(* IEC 61131-3 sources: Idecon_CheckWeigher_WP/03_FC, 6 files *)

(* ---- FC_Idecon_ResetBatch.st ---- *)
// ==============================================================================
// FUNZIONE: FC_Idecon_ResetBatch
// DESCRIZIONE: Resetta statistiche batch su cambio lotto
// INPUT: CurrentBatchCode (STRING[64]) - Codice lotto corrente
// OUTPUT: BatchResetDone (BOOL) - TRUE se reset eseguito
// NOTE: Implementare nel task ciclico monitorando cambio G_Idecon_BatchCode
// ==============================================================================

VAR_INPUT
    CurrentBatchCode : STRING[64];
END_VAR

VAR_OUTPUT
    BatchResetDone : BOOL;
END_VAR

VAR
    PreviousBatchCode : STRING[64];
    CurrentTimestamp_Unix_ms : LINT;
END_VAR

// Get current timestamp (requires SysTicks function or PLC time)
// CurrentTimestamp_Unix_ms := ...;  // Da implementare con funzione di sistema

// Detect batch code change
IF CurrentBatchCode <> PreviousBatchCode THEN
    // Reset all statistics
    G_Idecon_BatchStats.BatchStartTime_Unix := CurrentTimestamp_Unix_ms;
    G_Idecon_BatchStats.BatchDuration_Sec := 0;
    G_Idecon_BatchStats.TotalProducts := 0;
    G_Idecon_BatchStats.AcceptedProducts := 0;
    G_Idecon_BatchStats.RejectedUnderweight := 0;
    G_Idecon_BatchStats.RejectedOverweight := 0;
    G_Idecon_BatchStats.MissingProducts := 0;
    G_Idecon_BatchStats.TotalWeight_kg := 0.0;
    G_Idecon_BatchStats.AverageWeight_g := 0.0;
    G_Idecon_BatchStats.MinWeightMeasured_g := 999999.0;
    G_Idecon_BatchStats.MaxWeightMeasured_g := 0.0;
    G_Idecon_BatchStats.StdDeviation_g := 0.0;
    G_Idecon_BatchStats.YieldPercentage := 0.0;
    G_Idecon_BatchStats.RejectionRate := 0.0;
    G_Idecon_BatchStats.ProductionRate_PPM := 0.0;
    G_Idecon_BatchStats.BatchActive := TRUE;
    G_Idecon_BatchStats.DataValid := FALSE;

    // Save previous batch code
    PreviousBatchCode := CurrentBatchCode;

    BatchResetDone := TRUE;
ELSE
    BatchResetDone := FALSE;
END_IF;

// Update duration if batch is active
IF G_Idecon_BatchStats.BatchActive AND CurrentTimestamp_Unix_ms > 0 THEN
    G_Idecon_BatchStats.BatchDuration_Sec := (CurrentTimestamp_Unix_ms - G_Idecon_BatchStats.BatchStartTime_Unix) / 1000;
END_IF;

(* ---- FC_Idecon_UpdateBatchStats.st ---- *)
// ==============================================================================
// FUNZIONE: FC_Idecon_UpdateBatchStats
// DESCRIZIONE: Aggiorna statistiche batch su ogni pesata ricevuta da IDECON
// NOTE: Chiamare nel task ciclico quando G_Idecon_LastWeight.Valid = TRUE
// ==============================================================================

// Increment total counter
G_Idecon_BatchStats.TotalProducts := G_Idecon_BatchStats.TotalProducts + 1;

// Classify based on weight limits
IF G_Idecon_LastWeight.Weight_g >= G_Idecon_BatchConfig.MinWeight_g AND
   G_Idecon_LastWeight.Weight_g <= G_Idecon_BatchConfig.MaxWeight_g THEN
    G_Idecon_BatchStats.AcceptedProducts := G_Idecon_BatchStats.AcceptedProducts + 1;
ELSIF G_Idecon_LastWeight.Weight_g < G_Idecon_BatchConfig.MinWeight_g THEN
    G_Idecon_BatchStats.RejectedUnderweight := G_Idecon_BatchStats.RejectedUnderweight + 1;
ELSE
    G_Idecon_BatchStats.RejectedOverweight := G_Idecon_BatchStats.RejectedOverweight + 1;
END_IF;

// Update weight statistics
G_Idecon_BatchStats.TotalWeight_kg := G_Idecon_BatchStats.TotalWeight_kg + (G_Idecon_LastWeight.Weight_g / 1000.0);

// Update average weight
IF G_Idecon_BatchStats.TotalProducts > 0 THEN
    G_Idecon_BatchStats.AverageWeight_g := (G_Idecon_BatchStats.TotalWeight_kg * 1000.0) / TO_REAL(G_Idecon_BatchStats.TotalProducts);
END_IF;

// Update min/max measured
IF G_Idecon_LastWeight.Weight_g < G_Idecon_BatchStats.MinWeightMeasured_g OR
   G_Idecon_BatchStats.TotalProducts = 1 THEN
    G_Idecon_BatchStats.MinWeightMeasured_g := G_Idecon_LastWeight.Weight_g;
END_IF;

IF G_Idecon_LastWeight.Weight_g > G_Idecon_BatchStats.MaxWeightMeasured_g THEN
    G_Idecon_BatchStats.MaxWeightMeasured_g := G_Idecon_LastWeight.Weight_g;
END_IF;

// Calculate KPIs
IF G_Idecon_BatchStats.TotalProducts > 0 THEN
    G_Idecon_BatchStats.YieldPercentage := (TO_REAL(G_Idecon_BatchStats.AcceptedProducts) /
                                           TO_REAL(G_Idecon_BatchStats.TotalProducts)) * 100.0;
    G_Idecon_BatchStats.RejectionRate := (TO_REAL(G_Idecon_BatchStats.RejectedUnderweight +
                                                   G_Idecon_BatchStats.RejectedOverweight) /
                                           TO_REAL(G_Idecon_BatchStats.TotalProducts)) * 100.0;
END_IF;

// Calculate production rate (pieces per minute)
IF G_Idecon_BatchStats.BatchDuration_Sec > 0 THEN
    G_Idecon_BatchStats.ProductionRate_PPM := TO_REAL(G_Idecon_BatchStats.TotalProducts) /
                                               (TO_REAL(G_Idecon_BatchStats.BatchDuration_Sec) / 60.0);
END_IF;

// Set data valid flag after first product
IF G_Idecon_BatchStats.TotalProducts >= 1 THEN
    G_Idecon_BatchStats.DataValid := TRUE;
END_IF;

(* ---- IDECON_AsciiByteToChar.st ---- *)
// ==============================================================================
// FUNZIONE: IDECON_AsciiByteToChar
// DESCRIZIONE: Converte un Byte ASCII nel corrispondente carattere Stringa
// ==============================================================================

// Variabili Interne (Dichiarare in Sysmac):
// u : USINT

u := BYTE_TO_USINT(InByte);

CASE u OF
    16#20: IDECON_AsciiByteToChar := ' ';
    16#2D: IDECON_AsciiByteToChar := '-';
    16#2E: IDECON_AsciiByteToChar := '.';
    16#2F: IDECON_AsciiByteToChar := '/';
    16#3A: IDECON_AsciiByteToChar := ':';
    16#3D: IDECON_AsciiByteToChar := '=';
    16#3F: IDECON_AsciiByteToChar := '?';
    16#5F: IDECON_AsciiByteToChar := '_';
    16#7C: IDECON_AsciiByteToChar := '|';
    16#30: IDECON_AsciiByteToChar := '0';
    16#31: IDECON_AsciiByteToChar := '1';
    16#32: IDECON_AsciiByteToChar := '2';
    16#33: IDECON_AsciiByteToChar := '3';
    16#34: IDECON_AsciiByteToChar := '4';
    16#35: IDECON_AsciiByteToChar := '5';
    16#36: IDECON_AsciiByteToChar := '6';
    16#37: IDECON_AsciiByteToChar := '7';
    16#38: IDECON_AsciiByteToChar := '8';
    16#39: IDECON_AsciiByteToChar := '9';
    16#41: IDECON_AsciiByteToChar := 'A';
    16#42: IDECON_AsciiByteToChar := 'B';
    16#43: IDECON_AsciiByteToChar := 'C';
    16#44: IDECON_AsciiByteToChar := 'D';
    16#45: IDECON_AsciiByteToChar := 'E';
    16#46: IDECON_AsciiByteToChar := 'F';
    16#47: IDECON_AsciiByteToChar := 'G';
    16#48: IDECON_AsciiByteToChar := 'H';
    16#49: IDECON_AsciiByteToChar := 'I';
    16#4A: IDECON_AsciiByteToChar := 'J';
    16#4B: IDECON_AsciiByteToChar := 'K';
    16#4C: IDECON_AsciiByteToChar := 'L';
    16#4D: IDECON_AsciiByteToChar := 'M';
    16#4E: IDECON_AsciiByteToChar := 'N';
    16#4F: IDECON_AsciiByteToChar := 'O';
    16#50: IDECON_AsciiByteToChar := 'P';
    16#51: IDECON_AsciiByteToChar := 'Q';
    16#52: IDECON_AsciiByteToChar := 'R';
    16#53: IDECON_AsciiByteToChar := 'S';
    16#54: IDECON_AsciiByteToChar := 'T';
    16#55: IDECON_AsciiByteToChar := 'U';
    16#56: IDECON_AsciiByteToChar := 'V';
    16#57: IDECON_AsciiByteToChar := 'W';
    16#58: IDECON_AsciiByteToChar := 'X';
    16#59: IDECON_AsciiByteToChar := 'Y';
    16#5A: IDECON_AsciiByteToChar := 'Z';
    16#61: IDECON_AsciiByteToChar := 'a';
    16#62: IDECON_AsciiByteToChar := 'b';
    16#63: IDECON_AsciiByteToChar := 'c';
    16#64: IDECON_AsciiByteToChar := 'd';
    16#65: IDECON_AsciiByteToChar := 'e';
    16#66: IDECON_AsciiByteToChar := 'f';
    16#67: IDECON_AsciiByteToChar := 'g';
    16#68: IDECON_AsciiByteToChar := 'h';
    16#69: IDECON_AsciiByteToChar := 'i';
    16#6A: IDECON_AsciiByteToChar := 'j';
    16#6B: IDECON_AsciiByteToChar := 'k';
    16#6C: IDECON_AsciiByteToChar := 'l';
    16#6D: IDECON_AsciiByteToChar := 'm';
    16#6E: IDECON_AsciiByteToChar := 'n';
    16#6F: IDECON_AsciiByteToChar := 'o';
    16#70: IDECON_AsciiByteToChar := 'p';
    16#71: IDECON_AsciiByteToChar := 'q';
    16#72: IDECON_AsciiByteToChar := 'r';
    16#73: IDECON_AsciiByteToChar := 's';
    16#74: IDECON_AsciiByteToChar := 't';
    16#75: IDECON_AsciiByteToChar := 'u';
    16#76: IDECON_AsciiByteToChar := 'v';
    16#77: IDECON_AsciiByteToChar := 'w';
    16#78: IDECON_AsciiByteToChar := 'x';
    16#79: IDECON_AsciiByteToChar := 'y';
    16#7A: IDECON_AsciiByteToChar := 'z';
ELSE
    IDECON_AsciiByteToChar := '?';
END_CASE;

(* ---- IDECON_FieldAt.st ---- *)
// ==============================================================================
// FUNZIONE: IDECON_FieldAt
// DESCRIZIONE: Estrae un campo da una stringa separata da delimitatori (es. '|')
// NOTA CRITICA: Utilizza sintassi MID(Testo, Lunghezza, Posizione)
// ==============================================================================

// Variabili Interne (Dichiarare in Sysmac):
// i, n, startPos, endPos, curIndex, resultLen : UINT
// sCh : STRING[2]

n := LEN(InText);
startPos := 1;
endPos := 0;
curIndex := 0;

IF Index = 0 THEN
    IDECON_FieldAt := '';
    RETURN;
END_IF;

FOR i := 1 TO n DO
    sCh := MID(InText,1, i);
    IF sCh = Delim THEN
        curIndex := curIndex + 1;
        IF curIndex = Index THEN
            endPos := i - 1;
            EXIT;
        END_IF;
        startPos := i + 1;
    END_IF;
END_FOR;

IF endPos = 0 THEN
    curIndex := curIndex + 1;
    IF curIndex = Index THEN
        endPos := n;
    END_IF;
END_IF;

IF endPos < startPos THEN
    IDECON_FieldAt := '';
    RETURN;
END_IF;

resultLen := endPos - startPos + 1;
IDECON_FieldAt := MID(InText,  resultLen,startPos);

(* ---- IDECON_ParseHexDword.st ---- *)
// ==============================================================================
// FUNZIONE: IDECON_ParseHexDword
// DESCRIZIONE: Converte una stringa esadecimale (es. '0x80') in DWORD
// ==============================================================================

// Variabili Interne:
// i, n : UINT
// sCh : STRING[1]
// posUpper, posLower : INT
// v, d : DINT
v := 0;
n := LEN(InText);
i := 1;

// Skip '0x'
IF n >= 2 THEN
    IF (MID(InText, 2, 1) = '0x') OR (MID(InText, 2, 1) = '0X') THEN i := 3; END_IF;
END_IF;

WHILE i <= n DO
    // Estrai carattere corrente
    // Usiamo FIND su stringhe letterali che è supportato ovunque
    // Cerchiamo il carattere nella mappa Hex

    // Cerca in "0123456789ABCDEFabcdef"
    // Posizione: 1=0, 10=9, 11=A, 16=F, 17=a, 22=f

    // Nota: MID(Source, Len, Pos)
    // FIND(Source, Target) -> Ritorna 1-based index

    d := 0; // Reset valore cifra

    // Cerca 0-9
    posUpper := FIND('0123456789', MID(InText, 1, i));
    IF posUpper > 0 THEN
        d := INT_TO_DINT(posUpper - 1); // '0'->1->0, '9'->10->9
        v := (v * 16) + d;
    ELSE
        // Cerca A-F
        posUpper := FIND('ABCDEF', MID(InText, 1, i));
        IF posUpper > 0 THEN
            d := INT_TO_DINT(posUpper - 1) + 10; // 'A'->1->10
            v := (v * 16) + d;
        ELSE
            // Cerca a-f
            posLower := FIND('abcdef', MID(InText, 1, i));
            IF posLower > 0 THEN
                d := INT_TO_DINT(posLower - 1) + 10; // 'a'->1->10
                v := (v * 16) + d;
            END_IF;
        END_IF;
    END_IF;

    i := i + 1;
END_WHILE;

IDECON_ParseHexDword := DINT_TO_DWORD(v);

(* ---- IDECON_StartsWith.st ---- *)
// ==============================================================================
// FUNZIONE: IDECON_StartsWith
// DESCRIZIONE: Restituisce TRUE se InText inizia con Prefix
// ==============================================================================

// Variabili Interne:
// prefixLenU : UINT
// prefixLen, textLen : INT

prefixLenU := LEN(Prefix);
prefixLen := UINT_TO_INT(prefixLenU);
textLen := UINT_TO_INT(LEN(InText));

IF prefixLen <= 0 THEN
    IDECON_StartsWith := TRUE;
ELSIF textLen < prefixLen THEN
    IDECON_StartsWith := FALSE;
ELSE
	// Controlla "prefixLenU" caratteri a partire dalla posizione 1
    IDECON_StartsWith := (MID(InText,  prefixLenU,1) = Prefix);
END_IF;
